// =============================================================================
// 02_DataBlocks.scl
// All non-recipe data blocks.
// Recipe program DBs (DB_RecipeProgram1..10) are in 02b_RecipePrograms.scl.
// They live in LOAD memory; the machine runs from DB_SelectedRecipe (this file).
// Target: CPU 1214C (100KB work memory)
// =============================================================================

// -----------------------------------------------------------------------------
// DB_HMI - Human Machine Interface data
// -----------------------------------------------------------------------------
DATA_BLOCK "DB_HMI"
{ S7_Optimized_Access := 'TRUE' }
VERSION : 0.3
NON_RETAIN
    VAR
        // ===========================================================
        // BUTTONS (Input) - Version_GCODE compatible
        // ===========================================================
        Btn_Start : Bool;           // Start machine
        Btn_Stop : Bool;            // Stop machine
        Btn_Pause : Bool;           // Pause/Resume toggle
        Btn_Reset : Bool;           // Reset program to beginning
        Btn_ApplyToolConfig : Bool;  // Apply tool-slot codes from HMI to DB_ToolConfig
        Btn_AckError : Bool;        // Acknowledge error → transitions from STATE_ERROR to STOPPED
        Btn_Continue : Bool;        // Continue from pause (PAUSED) -- STATE_PAUSED → RUNNING
        Btn_Restart : Bool;         // STATE_ERROR or PAUSED → STOPPED (restart with Start)
        Btn_ProdReset : Bool;       // Reset production counters + history
        Btn_LastCycleReset : Bool;  // Reset last cycle summary only (counters preserved)
                                    // NOTE: Btn_ProdReset already does this too.
                                    // If not adding both as separate HMI buttons, Btn_LastCycleReset
                                    // is redundant -- do not connect to HMI if unused.

        // ===========================================================
        // MODE SELECTION (Input)
        // ===========================================================
        ProductSelect : Int := 1;           // Recipe selector (1-50) -- 50 slots since 2026-08-10 (was 10)
        FeedrateOverride : Real := 100.0;   // Speed % for G1 moves (50-200, 100=normal)
        RapidOverride : Real := 100.0;      // Speed % for G0 rapid moves (50-200)
        SingleStepMode : Bool := FALSE;     // TRUE = stop after each line, wait for StepNext
        StepNext : Bool := FALSE;           // Pulse to advance one step in SingleStepMode

        // Program names and validity.
        //
        // *** DELIBERATELY NOT EXTENDED TO 50 (2026-08-10). Read before touching. ***
        // Verified 2026-08-10: NOTHING in this project writes or reads either array --
        // not the PLC, and not the CAM post-processor (grep gcodes/ for ProgramNames:
        // no hits). They have been declared-and-unused since 1..5. At 50 slots they would
        // cost ~1.1 KB of the 100 KB work memory to stay just as unused, on a CPU that ran
        // out of work memory on 2026-07-31.
        //
        // The name problem is solved two other ways instead:
        //   - WHICH program is loaded now: DB_HMI.LoadedProgramName, a continuous mirror of
        //     DB_SelectedRecipe.Header.sName. One String[20] regardless of slot count.
        //   - BROWSING all 50 names before selection: a WinCC text list keyed off
        //     ProductSelect. Zero PLC bytes, and operator-editable on the HMI, which is what
        //     "operator-defined names" wanted in the first place.
        //
        // Kept at 1..10 rather than deleted because the WinCC project may write them and it
        // is not visible from here -- deleting would silently break an HMI tag connection.
        // If the HMI does not use them either, they are ~230 B of reclaimable work memory.
        ProgramNames : Array[1..10] of String[20];  // UNUSED -- see note above
        ProgramValid : Array[1..10] of Bool;        // UNUSED -- see note above

        // Name of the recipe currently in DB_SelectedRecipe (2026-08-10). PLC-written,
        // read-only for the HMI. Continuous mirror of DB_SelectedRecipe.Header.sName,
        // written at the bottom of FB_Process next to the DB_Diagnostic mirrors -- so it
        // appears in no reset path by design (nothing to clear; it always reports the
        // buffer's true content, blank when the buffer is poisoned or a load failed).
        // 22 bytes, flat regardless of slot count. Display it beside ProductSelect so the
        // operator sees WHICH program is about to run, not just a slot number out of 50.
        // NOTE: CAM currently emits the same generic sName ('SpinningCam Program') for
        // every program -- ask SpinningCam for a distinct name per program or this reads
        // identically for all 50 slots.
        LoadedProgramName : String[20];

        // Recipe checksum pair, PLC-written, read-only for the HMI (2026-08-14).
        // Continuous mirrors written next to LoadedProgramName at the bottom of
        // FB_Process -- in no reset path by design, because they always report the
        // buffer's true state. 9 bytes total.
        //
        // Display these two side by side on the diagnostics screen. They matter only
        // when they DISAGREE, and then they answer the one question 16#0316 cannot:
        // which side is wrong. Three implementations of the algorithm exist
        // (SpinningCam's, tools/split_recipe_db.py, FB_RecipeLoader) and only the
        // first two have ever been checked against each other. If _Calculated is a
        // stable, repeatable number that simply is not _Recipe, suspect the SCL, not
        // the recipe file -- re-exporting a good file will not help and wastes a trip.
        // If _Calculated changes between attempts on the same recipe, the transfer is
        // landing different data each time, which is the original fault.
        //
        // _Verified = TRUE means checked AND matched. FALSE also means "this recipe
        // carries no checksum", so it is not a fault indicator on its own -- a blank
        // _Recipe (0) with _Verified FALSE is a pre-2026-08-14 export loading normally.
        Checksum_Recipe : UDInt;        // what the recipe file declares
        Checksum_Calculated : UDInt;    // what the PLC computed after reassembly
        Checksum_Verified : Bool;       // TRUE = checked and matched


        // Tool slot codes editable from HMI. Enter external codes like 101, 406 etc.
        // These are copied to DB_ToolConfig.ToolCode_List when operator presses Apply.
        ToolSlotCode : Array[1..4] of Int := [101, 102, 103, 104];

        // ===========================================================
        // POSITION DISPLAYS (Output)
        // ===========================================================
        ActualX : Real;             // Current X position (mm)
        ActualZ : Real;             // Current Z position (mm)

        // ===========================================================
        // STATUS DISPLAYS (Output)
        // ===========================================================
        StatusMsg : String[50];     // Status message text
        MachineState : Int;         // State machine state
        CurrentLine : Int;          // Current line being executed
        TotalLines : Int;           // Total lines in program
        // -----------------------------------------------------------
        // Pass display -- mirrored from FB_RecipeHandler every scan.
        // Fed by the CMD=50 / CMD=51 marker lines SpinningCam emits when its
        // PLC-mode "pass markers" option is on. 0 = NO PASS INFORMATION (recipe
        // has no markers, or the first one has not been reached yet), so the HMI
        // must blank the whole group on 0 rather than display "Pass 0 / 0".
        // "Line 47 of 99" means nothing to an operator; "Op 1, pass 3 of 10" is
        // how the job is actually described. See letter_spinningcam_pass_markers.md.
        // -----------------------------------------------------------
        CurrentOp : Int;            // Operation number of the current line (0 = unknown)
        TotalOps : Int;             // Operations in the loaded program (0 = unknown)
        CurrentPass : Int;          // Pass number within the current operation (0 = unknown)
        TotalPasses : Int;          // Passes in the current operation (0 = unknown)
        ProgressPercent : Real;     // Progress 0-100%
        CurrentTool : Int;          // Active tool (1-4)
        FeedrateActive : Real;      // Actual feedrate (mm/min)
        // ⚠️ UNUSED: PLC code does not write to the Axis_Status_* tags below anywhere.
        // They will always be 0 / empty if connected to HMI. Reserved for future use
        // -- do not display on HMI for now.
        Axis_Status_X        : Int;
        Axis_Status_Z        : Int;
        Axis_Status_Spindle  : Int;
        Axis_Status_Toolhead : Int;
        Axis_Status_X_Str        : String[10];
        Axis_Status_Z_Str        : String[10];
        Axis_Status_Spindle_Str  : String[10];
        Axis_Status_Toolhead_Str : String[10];
        // ===========================================================
        // STATUS LAMPS (Output)
        // ===========================================================
        IsRunning : Bool;           // Machine is running
        IsPaused : Bool;            // Machine is paused
        HasError : Bool;            // Error is active
        ElapsedTime : Time;         // Program elapsed time
        ElapsedSeconds : DInt;      // Elapsed time in seconds (for HMI display)
        // CycleCount DELETED 2026-08-15 -- it duplicated "DB_Production".TotalOK and was
        // wrong (its one-shot only cleared on a hard reset, so it counted once per Reset
        // press, not once per part). Parts counting lives in DB_Production alone:
        // TotalStarted / TotalOK / TotalNOK / TotalStopped / TotalAborted. Do not add a
        // parts counter back into DB_HMI.

        // ===========================================================
        // ERROR DISPLAY (Output)
        // ===========================================================
        ErrorID : Word;             // Error code (0=OK)
        ErrorText : String[100];     // Error description
        ErrorDetail : String[120];   // Additional error info

        // ===========================================================
        // WARNING DISPLAY (Output)
        // ===========================================================
        HasWarning : Bool;          // TRUE when a non-blocking warning is active (E-Stop bypass or sheet insert prompt)
        // Key for the HMI's warning text list (ITEM-55). Written every scan next to
        // WarningText, so it needs no reset-path entry: the ELSE branch of the warning
        // block drives it to 0 unconditionally. 0 must stay "no warning".
        //   1 = DANGER: E-Stop bypassed - machine runs unguarded (auto run IS permitted
        //       since 2026-08-12 -- this is the only on-screen sign of it)
        //   2 = Insert sheet, then press both start buttons
        //   3 = Tool axis locked - ToolHeadLock is engaged (manual jog/move/home
        //       on the tool axis refused; see the interlock in FB_Process)
        WarningID : Int;
        WarningText : String[70];   // Warning message text -- English (E-Stop bypass or operator prompts only)
        ResumeLine : Int := -1;     // Saved recipe line for warm restart (-1 = none). Set in STATE_ERROR, cleared on Btn_Restart.

        // End-of-program sanding dwell in progress (2026-08-29). PLC-written, read-only
        // for the HMI. TRUE = the program has finished AND the spindle has been deliberately
        // restarted at DB_MachineConfig.SandSpeed so the operator can sand the part.
        //
        // Display this prominently. MachineState is 100 ('Program Complete') throughout the
        // dwell, so without this flag the screen says the machine is finished while the
        // spindle is turning -- which is exactly the moment an operator reaches in.
        // It is the key for the sanding banner in the WinCC text lists; MachineState cannot
        // serve, because it does not change when the dwell starts or ends.
        //
        // No reset-path entry needed: it is a continuous mirror of the FB_Process latch,
        // written every scan next to the DB_Diagnostic mirrors at the bottom of FB_Process,
        // so it follows the latch to FALSE on every exit path.
        SandActive : Bool;

        // ===========================================================
        // SPANISH TEXT MIRRORS -- REMOVED 2026-08-10 (ITEM-55, stage 1).
        // StatusMsg_ES / ErrorText_ES / ErrorDetail_ES / WarningText_ES are gone,
        // along with the 161 PLC assignments that filled them (~4.9 KB of string
        // literals plus the copy code, on a CPU that hit 101% work memory).
        // Spanish now comes from WinCC text lists keyed off tags the PLC already
        // writes: ErrorID, MachineState, DB_Manual.MDI_Status, and WarningID.
        // The wording was extracted to tools/hmi_texts.csv BEFORE deletion -- use
        // that to populate the text lists; do not retype or re-translate.
        // Do NOT re-add per-language string fields here: each new language then
        // costs work memory again, which is exactly what this removed.
        // ===========================================================

        // ===========================================================
        // BYPASS SWITCHES (for testing) - Version_GCODE compatible
        // ⚠️ All bypasses reset to FALSE on restart (FC_LoadConfig).
        // All must be FALSE in production.
        // ===========================================================
        // ⚠️ Bypass_EStop PERMITS AUTO RUN since 2026-08-12 (it used to block it).
        // The machine will execute a recipe with the E-Stop circuit defeated.
        // Protect this tag with a WinCC user authorization (service login only) --
        // the PLC deliberately no longer second-guesses it. Still forced FALSE by
        // FC_LoadConfig on every power-up, so it cannot survive a restart.
        Bypass_EStop        : Bool := FALSE;  // Used in FB_SafetyMonitor ✅
        Bypass_Door         : Bool := TRUE;  // Used in FB_SafetyMonitor ✅
        Bypass_AirPressure  : Bool := TRUE;  // Used in FB_SafetyMonitor ✅
        Bypass_Drives       : Bool := FALSE;  // Used in FB_SafetyMonitor ✅
        Bypass_Spindle      : Bool := FALSE;  // Skips spindle commands in recipe (FB_RecipeHandler) -- dry run / commissioning
        Bypass_ToolChanger  : Bool := FALSE;  // ⚠️ UNUSED -- not in safety monitor
        // Bypass_MandrelLock DELETED from DB_HMI 2026-08-16 -- it was an ORPHAN. ITEM-33 declared
        // it here as well as in DB_MachineConfig, but every one of the nine read sites, and
        // FC_LoadConfig, use "DB_MachineConfig".Bypass_MandrelLock. This copy was written by
        // nothing and read by nothing. Two identically-named flags where only one is live is a
        // trap: an HMI switch bound to this one would appear to bypass the cylinder and do
        // absolutely nothing. The live flag is DB_MachineConfig.Bypass_MandrelLock -- use that.
        Bypass_ToolHeadLock : Bool := FALSE;  // TRUE = skip ToolHeadLock sensor wait in STATE_LOCK_EXTEND_WAIT (no cylinder/sensor); cylinder still commanded if present
        // A Sim_HomeInPlace flag was added here on 2026-09-06 and REVERTED the same day.
        // It selected MC_Home Mode 0 so a homing cycle could finish in PLCSIM. It cannot
        // work: S7-PLCSIM does not simulate S7-1200 motion control at all -- the
        // technology objects download, but their logic never runs and the PTO hardware is
        // not simulated -- so MC_Power never reports Status and MC_Home never completes,
        // in any mode. Do not re-add it. Nothing past STATE_STARTING can be simulated;
        // what CAN be tested offline is everything before it (recipe load, checksum,
        // pre-scan). See CLAUDE.md and the PLCSIM section of Human_TODO.md.

        // ===========================================================
        // BOUNDING BOX (Output - from pre-scan)
        // ===========================================================
        BoundingBox_MinX : Real;
        BoundingBox_MaxX : Real;
        BoundingBox_MinZ : Real;
        BoundingBox_MaxZ : Real;
        BoundingBox_Valid : Bool;
        PreScanProgress : Real := 0.0;  // Pre-scan progress 0-100% (written during STATE_PRE_SCAN)

        // ===========================================================
        // MANUAL > MANAGE: Contactor & Enable controls (Input)
        // HMI writes these; PLC drives physical outputs in OB1.
        // Buttons are toggles (maintained, not momentary).
        // ===========================================================
        Btn_Contactor_X       : Bool;   // Energize X driver contactor
        Btn_Contactor_Z       : Bool;   // Energize Z driver contactor
        Btn_Contactor_Tool    : Bool;   // Energize Tool driver contactor
        Btn_Contactor_Spindle : Bool;   // Energize Spindle driver contactor
        Btn_Enable_X          : Bool;   // Send enable signal to X drive
        Btn_Enable_Z          : Bool;   // Send enable signal to Z drive
        // Btn_Enable_Tool (2026-08-16): treated exactly like Btn_Enable_X/Z -- an HMI toggle on
        // MANUAL > MANAGE, ALSO forced TRUE by STATE_STARTING on every auto start. Same drive
        // model, same treatment, no settle delay, no bypass term (FC_ContactorControl ANDs the
        // output with Btn_Contactor_Tool). Before this the tool had no enable output at all:
        // the drive's enable was linked on locally, so the servo came up enabled the instant its
        // contactor closed. The wire is now landed on %Q8.1 and that link is removed.
        Btn_Enable_Tool       : Bool;   // Send enable signal to Tool drive

        // MANUAL > MANAGE: Status feedback (Output) for HMI lamps
        // PLC writes these back after applying safety interlock.
        Contactor_X_On       : Bool;
        Contactor_Z_On       : Bool;
        Contactor_Tool_On    : Bool;
        Contactor_Spindle_On : Bool;
        Enable_X_On          : Bool;
        Enable_Z_On          : Bool;
        Enable_Tool_On       : Bool;

        // ===========================================================
        // E-STOP DUAL CHANNEL STATUS (Output - PLC writes, HMI reads)
        // ===========================================================
        EStop_Ch1_OK      : Bool;   // Channel 1 contact state (TRUE=closed=safe)
        EStop_Ch2_OK      : Bool;   // Channel 2 contact state (TRUE=closed=safe)
        EStop_Discrepancy : Bool;   // Ch1 ≠ Ch2 → contact fault, service required
    END_VAR
BEGIN
END_DATA_BLOCK

// -----------------------------------------------------------------------------
// DB_MachineConfig - Machine configuration parameters
//
// RETENTIVITY (changed 2026-08-09) -- NON_RETAIN was REMOVED from this block.
//
// Why: the commissioning values the operator types on the HMI and that FC_LoadConfig
// deliberately does NOT rewrite -- SheetLoadPos_X, SheetLoadPos_Z, SheetLoadTol -- were
// lost on every power cycle. A non-retentive DB is re-initialised from its start values
// in load memory on restart, so the machine came back parking at 200.0 / 170.0 no matter
// what was set on the HMI.
//
// MANUAL STEP REQUIRED IN TIA PORTAL AFTER IMPORTING THIS SOURCE:
//   Open DB_MachineConfig and tick "Retain" on -- at minimum --
//       SheetLoadPos_X, SheetLoadPos_Z, SheetLoadTol, SandTime_s, SandSpeed
//   The other operator-owned values have the same problem and are worth ticking too:
//       SoftLimit_MinX/MaxX/MinZ/MaxZ, SafePos_X/Z, PauseRetract_X/Z/Vel,
//       HomeOffset_X/Z
//   Source import cannot set per-tag retentivity; removing NON_RETAIN only makes the
//   checkbox available. VERIFY the checkboxes after every re-import of this file.
//
//   Do NOT tick Retain on anything FC_LoadConfig writes -- OB100 overwrites it on every
//   restart, so Retain has no effect there and only consumes retentive memory. That is
//   the whole "FIXED" section below, plus these four from the HMI-editable group:
//       HomeVelocity, PostHome_Clearance, AlwaysHomeOnAutoStart, and DB_Manual.HomingMode
//
// NOTE: changing retentivity forces a full re-initialisation of this DB on the next
// download (values return to the start values below). Re-enter the park position on the
// HMI once after that download.
// -----------------------------------------------------------------------------
DATA_BLOCK "DB_MachineConfig"
{ S7_Optimized_Access := 'TRUE' }
VERSION : 0.3
    VAR
        // =====================================================================
        // HMI-EDITABLE: Machine Physical Limits (mm)
        // These values are NOT overwritten by FC_LoadConfig.
        // Can be changed from HMI Setup screen. They survive a PLC restart ONLY if the
        // tag is marked Retain in the TIA DB editor -- see the block header.
        // =====================================================================
        SoftLimit_MinX : Real := -30.0;     // X minimum (home=0)
        SoftLimit_MaxX : Real := 500.0;   // X maximum travel (mm)
        SoftLimit_MinZ : Real := -50.0;  // Z minimum (negative = mandrel front / clearance)
        SoftLimit_MaxZ : Real := 500.0;   // Z maximum (forming depth)

        // HMI-EDITABLE: Safe Positions (mm)
        SafePos_X : Real := 0.0;         // "Go Safe" X target
        SafePos_Z : Real := 0.0;        // "Go Safe" Z target (clearance zone)

        // HMI-EDITABLE: Sheet-Load Park Position (mm)
        // The single position the machine parks at whenever it is waiting for the
        // operator to load a sheet. Reached at the end of every program (STATE_COMPLETE
        // is not used -- the park move is the STOPPING/POST_HOME_CLR path), after every
        // homing cycle, and after a Stop. STATE_STARTING compares the live axis position
        // against it to decide whether the homing seek can be skipped (fast cycle mode).
        //
        // SAFETY: this is where the operator reaches in to insert a sheet and where the
        // MandrelLock clamps. Set it only to a position where the tool head does not
        // obstruct loading. Commission conservatively (near 0,0) and walk it in.
        // Targets are clamped to SoftLimit_Min/Max before any move is issued.
        //
        // Deliberately NOT written by FC_LoadConfig, so OB100 does not fight the HMI.
        // MUST be marked Retain in the TIA DB editor -- see the block header. Without the
        // Retain tick these three revert to the start values below on every power cycle.
        SheetLoadPos_X : Real := 200.0;    // Sheet-load park X target (mm)
        SheetLoadPos_Z : Real := 170.0;    // Sheet-load park Z target (mm)
        SheetLoadTol   : Real := 2.0;    // +/- window counted as "at the park position" (mm)

        // HMI-EDITABLE: Pause Retract (mm / mm/s)
        // On Pause, X and Z jog by these signed offsets to pull the tool clear
        // (spindle keeps running). On Continue they return to the exact interruption
        // point before the recipe resumes. Retract target is clamped to soft limits.
        // Offset 0 = that axis does not move on pause. See docs/FB_Process_States.md
        // (STATE_PAUSED) for the full pause/resume sequence.
        PauseRetract_X   : Real := -10.0;   // Pause retract offset X (signed, mm)
        PauseRetract_Z   : Real := -10.0;   // Pause retract offset Z (signed, mm)
        PauseRetract_Vel : Real := 20.0;    // Retract/return velocity (mm/s)

        // HMI-EDITABLE: Homing Parameters
        HomeOffset_X : Real := 0.0;       // X set value after homing
        HomeOffset_Z : Real := 0.0;       // Z set value after homing
        HomeVelocity : Real := 10.0;      // Homing clearance velocity (mm/s)
        PostHome_Clearance : Real := 10.0; // Distance to clear PNP zone after homing (mm)
        // HMI-EDITABLE: fast cycle mode master switch.
        //   TRUE  = home all axes on every auto start (legacy behaviour)
        //   FALSE = skip the reference seek when the reference is trusted AND the axes
        //           are parked at SheetLoadPos (see FB_Process STATE_STARTING)
        // This switch can only ever skip homing in the NORMAL case. It never overrides
        // FB_Process bRequireHoming -- an E-Stop, a fault or a power-up always re-homes.
        AlwaysHomeOnAutoStart : Bool := FALSE;

        // ⚠️ UNUSED: The following two parameters are not read anywhere in PLC code.
        // Recipe handler takes its own feedrate from the recipe line.
        // Do not connect to HMI. May be used if manual tool change sequence is added later.
        ToolChangePos_X : Real := 0.0;   // (Unused) Safe X for manual tool change
        ToolChangePos_Z : Real := 0.0;  // (Unused) Safe Z for manual tool change
        DefaultFeedrate : Real := 100.0;  // (Unused) Default feedrate

        // =====================================================================
        // FIXED: Hardware/TO Limits -- must not be changed from HMI
        // FC_LoadConfig (OB100) writes these values on every restart.
        // =====================================================================
        MaxVelocity : Real := 40.0;     // mm/s - TO max velocity
        RapidVelocity : Real := 40.0;   // mm/s - G0 rapid speed
        MinVelocity : Real := 1.0;      // mm/s - TO minimum
        FeedrateConvFactor : Real := 60.0; // divisor to convert recipe F (mm/min) to axis velocity (mm/s)

        // EXPERIMENTAL -- velocity-mode continuous path (branch exp/velocity-path-350).
        // VelPath_Enable and VelPath_LeadTime are written by FC_LoadConfig on every
        // restart, so an online change lasts until the next power cycle. VelPath_Enable
        // is forced FALSE there -- the experiment must be switched on deliberately.
        // VelPath_MaxDeviation is OPERATOR-OWNED (2026-09-16): HMI-editable, NOT written
        // by FC_LoadConfig, needs a manual Retain tick (docs/RETAINED_TAGS.md). Without
        // the tick it falls back to the start value below at power-up.
        // Design and test plan: docs/MotionSmoothing.md section 9.
        VelPath_Enable       : Bool := TRUE; // TRUE = runs of G1 lines use MC_MoveVelocity (no stop per line)
        VelPath_LeadTime     : Real := 0.09;   // s -- next line takes over at feed x this before the end point (capped at half the segment). Tuned with the jerk-aware sim (scan 45 ms, t1 0.06)
        VelPath_MaxDeviation : Real := 2.0;   // mm -- HMI-EDITABLE. Start value raised 1.0 -> 2.0 on 2026-09-21 (user). Off-path / backwards distance that faults with 16#000F. PLC clamps to 0.05..5.0 (VM_MAXDEV_MIN/MAX in 05_RecipeHandler.scl -- the clamped value is what the fault text prints). Above 0.8 mm (the final-pass roller-mandrel gap = sheet thickness) it no longer protects the mandrel

        // Tool Configuration -- HMI-EDITABLE: active slot count (1-4)
        ToolCount    : Int  := 3;
        ToolVelocity : Real := 50.0;   // deg/s -- turret rotation speed (clamped by TO max)

        // Hardware configuration -- set TRUE if this axis is not physically connected to the machine
        // (different from HMI bypasses: this is a hardware presence flag)
        Bypass_ToolAxis : Bool := FALSE;
        // THE live MandrelLock bypass -- all nine read sites and FC_LoadConfig use this one.
        // (A duplicate in DB_HMI was deleted 2026-08-16; it was never read.)
        // TRUE = no MandrelLock cylinder, sheet clamped manually. FC_LoadConfig sets the
        // per-machine value on every power-up and overrides this start value -- change it there,
        // not here. On THIS machine it is TRUE.
        Bypass_MandrelLock : Bool := FALSE;
        // Spindle deceleration wait: time between RunCmd=FALSE and next RunCmd=TRUE.
        // Set to match VFD deceleration ramp time. HMI-editable.
        SpindleDecelTime : Time := T#2S;
        // Pause resume spin-up wait: on Continue from PAUSED, the spindle is
        // restarted and this time is allowed for it to ramp back up to speed
        // BEFORE the axes return to the interruption point and machining resumes.
        // The axes stay clear of the workpiece (held at the pause-retract position)
        // for this whole window. Set to the measured VFD ramp-up time + margin.
        SpindleResumeSpeedupTime : Time := T#5S;
        // Load-memory recipe copy (FB_RecipeLoader, STATE_RECIPE_LOAD(11)):
        // hang watchdog on the READ_DBL transfer. A 1000-line recipe is ~12 KB
        // and completes in well under a second; this only catches a transfer
        // that never reports BUSY=FALSE. Expiry -> 16#0312, machine goes to
        // STATE_ERROR rather than starting a cycle on a half-copied recipe.
        RecipeLoadTimeout : Time := T#10S;
        // In-place spindle speed change (FB_SpindleControl): how long MC_MoveVelocity
        // Execute is held LOW to regenerate the trigger edge for the new velocity.
        // RunForward (VFD run) stays TRUE throughout -- only the PTO command edge is
        // regenerated. T#0S = one PLC scan. Increase if the VFD needs more settle
        // time before the new velocity command. Tune on-site.
        SpindleSpeedChange_ExecLowTime : Time := T#0S;
        // Speed-change mode selector (VFD-dependent -- confirm on the bench):
        //   FALSE = keep RunForward TRUE during the change (VFD tracks pulse-train
        //           frequency live; this is the documented wiring intent).
        //   TRUE  = also drop RunForward during the Execute-low window, then re-assert
        //           it. Use only if the drive latches its frequency at the RunForward
        //           rising edge and ignores a live frequency change. Safe re: PTO --
        //           the pulse train keeps running; RunForward is the stop signal.
        SpindleSpeedChange_DropRunForward : Bool := FALSE;
        // Proportional MandrelLock release wait (ITEM-28).
        // SpindleStopSafeTime = full-speed stop safety margin (tune to measured VFD decel time + margin).
        // Formula: PT = (capturedRPM / SpindleMaxRPM) * SpindleStopSafeTime
        // NOT a speed limit -- the only spindle limit is DB_Spindle.MaxSpeed (3000). This is the
        // denominator that scales the coast-down wait, and 2400 is deliberately BELOW it:
        // a smaller denominator makes PT longer, so the MandrelLock waits a little more than
        // strictly needed before releasing. Do NOT "sync" this to DB_Spindle.MaxSpeed -- raising
        // it to 3000 SHORTENS a safety wait. (An older comment here said "match
        // DB_Spindle.MaxSpeed"; that was misleading and is why this note exists. 2026-08-16.)
        SpindleMaxRPM       : Real := 2400.0;  // RPM -- denominator for the proportional wait only
        SpindleStopSafeTime : Time := T#20S;   // Full-speed decel safety margin (tune on-site)

        // ─── HMI-EDITABLE: End-of-program sanding dwell (2026-08-29)
        // After a program finishes, STATE_COMPLETE(100) restarts the spindle at SandSpeed
        // and holds it for SandTime_s seconds so the operator can sand the part before removing it.
        //
        // WHY IT IS A RESTART AND NOT A "KEEP RUNNING": by the time the machine reaches
        // STATE_COMPLETE the spindle is already fully stopped, and it cannot be otherwise.
        // The CAM emits CMD=21 (Spindle OFF) as the second-to-last recipe line, and
        // FB_RecipeHandler STATE_SPINDLE_STOP_WAIT(58) BLOCKS on DB_Spindle.IsRunning=FALSE
        // before it will advance to the CMD=99 END marker. So the dwell necessarily begins
        // after a stop, and costs the VFD's ramp-down + ramp-up (~2 s) before the part turns
        // again. Do not "optimise" that away by suppressing the final CMD=21 -- a recipe has
        // several CMD=21 lines (program 1 has four: 51, 60, 69, 70) and picking the right one
        // needs a pre-scan pass whose failure mode is a spindle left running.
        //
        // BOTH must be > 0 for the dwell to arm. SandTime_s := 0 (the download default)
        // is the OFF switch and leaves end-of-program behaviour exactly as it was.
        //
        // UNITS: SandTime_s is WHOLE SECONDS as a plain Int -- deliberately NOT the Time
        // type every other timer in this DB uses. An S7 Time is milliseconds underneath,
        // so an operator typing "10" into a numeric field would get 10 ms and conclude the
        // feature is broken. The other timers are commissioning values a technician sets
        // once from the TIA editor; this one is retyped at the machine per job, so the
        // units have to survive a plain number field. FB_Process clamps it to
        // 0..SAND_TIME_MAX_S (600 s) and converts to a Time PT.
        //
        // SAFETY: this is the one feature that invites a hand near a turning part. The door
        // interlock does NOT protect it -- FC_LoadConfig forces Bypass_Door := TRUE on every
        // power-up on this machine. What does stop it: E-Stop (drops bDrivesEnable, which is
        // FB_SpindleControl's Enable) and the Stop button (STATE_COMPLETE is excluded from
        // the STOPPING path, so Stop goes straight to STOPPED and STOPPED clears the spindle).
        // Commission SandSpeed LOW -- it is a hand-sanding speed, not a cutting speed.
        //
        // Deliberately NOT written by FC_LoadConfig, so OB100 does not fight the HMI.
        // MUST be marked Retain in the TIA DB editor -- see the block header. Without the
        // Retain tick these two revert to the start values below on every power cycle.
        SandTime_s : Int  := 0;        // SECONDS. 0 = feature off. Spindle run time at end of program. Clamped 0..600.
        SandSpeed  : Real := 0.0;      // RPM during the dwell. Clamped to DB_Spindle.MinSpeed/MaxSpeed.

        // ─── Cylinder stroke wait times (open-loop: tuned to physical stroke duration)
        // These are deliberate waits with no sensor feedback. Set slightly above measured stroke time.
        CylMandrelLock_ClampTime    : Time := T#5S;    // STATE_SHEET_WAIT ph.2: MandrelLock clamp stroke
        CylSheetHolder_RetractTime  : Time := T#5S;    // STATE_SHEET_WAIT ph.3: SheetHolder retract stroke
        CylToolHeadLock_PreDelay    : Time := T#1S;    // STATE_LOCK_EXTEND_WAIT: pre-delay before solenoid energises
        CylToolHeadLock_RetractTime : Time := T#3S;    // STATE_LOCK_RETRACT_WAIT: spring-return wait (no sensor)
        CylBackSupport_EndRetractTime : Time := T#2S;  // End-of-recipe BackSupport retract: Sol_B held this long, then all coils off

        // ─── Process timeouts (trigger errors when limits exceeded)
        Timeout_DriveReady     : Time := T#3S;     // STATE_STARTING: drives not ready within this time → error
        // NOTE: there is deliberately no tool-enable settle delay. The tool servo is the same
        // drive as X and Z, which assert enable in the same scan as their contactor and have
        // always worked. See STATE_STARTING in 06_MainProcess.scl.
        Timeout_Homing         : Time := T#120S;   // STATE_HOMING + STATE_STOP_GOHOME combined timeout
        Timeout_Motion         : Time := T#300S;   // Per-line G0/G1 motion timeout in FB_RecipeHandler
        Timeout_SpindleAtSpeed : Time := T#10S;    // CMD=20: spindle must reach target speed within this time
        Timeout_SpindleStop    : Time := T#15S;    // CMD=21: spindle must reach zero within this time
        Timeout_ToolChange     : Time := T#30S;    // Turret rotation must complete within this time
        Timeout_EStopDiscrep   : Time := T#500MS;  // E-Stop dual-channel discrepancy debounce
    END_VAR
BEGIN
END_DATA_BLOCK

// DB_ErrorCodes removed -- error codes are used as inline hex constants.
// Severity: 0=info, 1=warn, 2=error, 3=fatal

// -----------------------------------------------------------------------------
// DB_Error - Centralized error snapshot for debugging (non-invasive to HMI)
// -----------------------------------------------------------------------------
DATA_BLOCK "DB_Error"
{ S7_Optimized_Access := 'TRUE' }
VERSION : 0.1
NON_RETAIN
    VAR
        Active    : Bool := FALSE;       // TRUE when an active error is present
        Code      : Word := 0;           // Error code (matches DB_ErrorCodes)
        Severity  : Byte := 0;           // Priority tier: 1=warning, 2=project, 3=motion/TO, 4=safety (higher preempts lower on HMI display)
        Source    : String[20];          // Originating FB or category (e.g. 'Recipe', 'Safety')
        Line      : Int := -1;           // Recipe line (if applicable) or -1
        TimeStamp : DTL;                 // Timestamp captured with RD_SYS_T
        Details   : String[120];          // Free text details / ActiveErrorText
        // History ring buffer (last 10 errors) for post-mortem analysis
        History_Code    : Array[1..10] of Word;
        History_Time    : Array[1..10] of DTL;
        History_Source  : Array[1..10] of String[20];
        // String[40] (was String[80], 2026-07-31 memory reclaim -- saves 400 B).
        // Matches AlarmEntry.ErrorText[40] in DB_AlarmHistory, so both history views
        // truncate identically. Written via LEFT(..., 40) in FB_AlarmManager.
        History_Details : Array[1..10] of String[40];
        History_Index   : Int := 0;      // 1..10
        History_Count   : Int := 0;      // Number of valid entries (<=10)
        TotalErrorCount : DInt := 0;     // Lifetime error count (incremented on each new error)
    END_VAR
BEGIN
END_DATA_BLOCK

// -----------------------------------------------------------------------------
// DB_ToolConfig - Tool changer configuration
// -----------------------------------------------------------------------------
DATA_BLOCK "DB_ToolConfig"
{ S7_Optimized_Access := 'TRUE' }
VERSION : 0.2
NON_RETAIN
    VAR
        // Slot angles -- automatically calculated by FC_ToolAngleCalc (AutoCalcAngles=TRUE)
        // or manually entered from HMI Tool page (AutoCalcAngles=FALSE).
        // Machine has 3 physical slots: 0 / 120 / 240 deg. Slot 4 is unused (ToolCount=3).
        Tool1_Position : Real := 0.0;     // Slot 1 angle (degrees)
        Tool2_Position : Real := 120.0;   // Slot 2 angle (degrees)
        Tool3_Position : Real := 240.0;   // Slot 3 angle (degrees)
        Tool4_Position : Real := 0.0;     // Slot 4 unused (ToolCount=3)

        // Slot code mapping -- can be entered from HMI Tool page.
        // Operator enters which head code is in which slot.
        ToolCode_List : Array[1..4] of Int := [101, 102, 103, 104];

        CurrentTool : Int := 1;           // Active slot number (1-4)

        // HMI Tool page: automatic angle calculation
        // TRUE = calculate evenly spaced based on ToolCount (3 slots → 0/120/240)
        // FALSE = Tool1..4_Position open for manual entry
        AutoCalcAngles : Bool := TRUE;

        // Calculated step angle -- displayed on HMI for information (e.g. "90°/slot")
        ToolStepAngle_Calc : Real := 120.0;
    END_VAR
BEGIN
END_DATA_BLOCK

// -----------------------------------------------------------------------------
// DB_Spindle - Spindle configuration and status
// -----------------------------------------------------------------------------
DATA_BLOCK "DB_Spindle"
{ S7_Optimized_Access := 'TRUE' }
VERSION : 0.2
NON_RETAIN
    VAR
        // Configuration
        MinSpeed : Real := 120.0;         // Minimum spindle speed (RPM)
        MaxSpeed : Real := 3000.0;        // Maximum spindle speed (RPM)
        DefaultSpeed : Real := 1200.0;    // Default spindle speed (RPM)
        SpeedTolerance : Real := 5.0;     // Speed tolerance for AtSpeed (%)
        Bypass_AtSpeed : Bool := FALSE;   // TRUE = skip AtSpeed wait (use during commissioning without drive)

        // Commands (input from HMI/Program)
        Cmd_SetSpeed : Real;              // Commanded speed
        Cmd_Direction : Int;              // 1=CW, -1=CCW
        SpeedOverride : Real := 100.0;    // Speed override (%)

        // Status (output)
        IsRunning : Bool := FALSE;
        AtSpeed : Bool := FALSE;
        ActualSpeed : Real := 0.0;
        CommandedSpeed : Real := 0.0;
        Error : Bool := FALSE;
        ErrorID : Word := 0;

        // =====================================================================
        // DIAGNOSTICS -- written every scan; read from HMI watch table
        // Use these to trace the spindle start chain without TIA Portal online.
        // Chain:  ReqStart → bSpindleStart → StartInput → PrevStart → StartEdge → state
        // =====================================================================
        Diag_SpindleState  : Int;   // FB_SpindleControl state (0=Idle, 10=Starting, 20=Running, 30=Stopping, 999=Error)
        Diag_StartInput    : Bool;  // Actual Start pin arriving at FB_SpindleControl (Manual OR bSpindleStart)
        Diag_StopInput     : Bool;  // Actual Stop pin arriving at FB_SpindleControl
        Diag_EnableInput   : Bool;  // Actual Enable pin (bDrivesEnable)
        Diag_StartEdge     : Bool;  // Rising edge computed inside FB_SpindleControl (TRUE = spindle command accepted)
        Diag_PrevStart     : Bool;  // prevStart latch inside FB_SpindleControl (must go FALSE between starts)
        Diag_bSpindleStart : Bool;  // FB_Process internal flag bSpindleStart (set by recipe or RUNNING state)
        Diag_bSpindleStop  : Bool;  // FB_Process internal flag bSpindleStop
        Diag_ReqStart      : Bool;
        Diag_ReqStop       : Bool;
        Diag_MoveVelBusy   : Bool;  // MC_MoveVelocity.Busy   -- TO is processing the velocity command
        Diag_MoveVelInVel  : Bool;  // MC_MoveVelocity.InVelocity -- motor reached commanded speed

        // =====================================================================
        // HISTORY RING BUFFER -- last 20 state-change snapshots
        // A new entry is pushed whenever SpindleState, PrevStart, ReqStart or
        // StartEdge changes, capturing every meaningful transition in sequence.
        //
        // How to read:
        //   1. Hist_Count tells you how many valid entries exist (0..20).
        //   2. Hist_Head-1 (mod 20) is the MOST RECENT entry.
        //   3. Entries are indexed [0..19]; read them in Seq order.
        //   4. Write Hist_Clear := TRUE from HMI to wipe and start fresh.
        // =====================================================================
        Hist_Head  : Int := 0;          // Next write position (0..19, wraps)
        Hist_Count : Int := 0;          // Number of valid entries (0..20)
        Hist_SeqNum : Int := 0;         // Rolling sequence counter
        Hist_Clear  : Bool := FALSE;    // HMI: write TRUE to clear buffer (auto-resets)
        Hist_Log   : Array[0..19] of "UDT_SpindleSnap";
    END_VAR
BEGIN
END_DATA_BLOCK

// -----------------------------------------------------------------------------
// DB_Diagnostic - Runtime diagnostics and debugging
// -----------------------------------------------------------------------------
DATA_BLOCK "DB_Diagnostic"
{ S7_Optimized_Access := 'TRUE' }
VERSION : 0.1
NON_RETAIN
    VAR
        // =========================================================
        // PROCESS STATE
        // =========================================================
        Process_State : Int;
        Process_SafeToRun : Bool;
        Process_DrivesEnable : Bool;

        // =========================================================
        // RECIPE HANDLER STATE
        // =========================================================
        Recipe_CurrentProgram : Int;    // Active program number (1-50)
        // Which recipe is actually sitting in DB_SelectedRecipe (0 = none/invalid).
        // Written by STATE_RECIPE_LOAD(11) after a successful READ_DBL copy.
        // Diagnostic value: if this disagrees with Recipe_CurrentProgram, the
        // buffer is stale and the machine would be cutting the wrong geometry.
        Recipe_LoadedProgram : Int;
        Recipe_CurrentLine : Int;       // Current line being executed
        Recipe_TotalLines : Int;        // Total lines in program
        Recipe_TargetX : Real;          // Current target X
        Recipe_TargetZ : Real;          // Current target Z
        Recipe_Velocity : Real;         // Current velocity
        // Pre-scan results
        PreScan_Complete : Bool;
        PreScan_Valid : Bool;           // No limit violations found
        PreScan_ErrorLine : Int;        // Line with limit error (-1 if none)

        // =========================================================
        // MOVE STATUS
        // =========================================================
        MoveX_Busy : Bool;
        MoveX_Done : Bool;
        MoveX_Error : Bool;
        MoveZ_Busy : Bool;
        MoveZ_Done : Bool;
        MoveZ_Error : Bool;
        bMoveX : Bool;                  // X axis needs to move
        bMoveZ : Bool;                  // Z axis needs to move

        // =========================================================
        // AXIS INFO (commissioning)
        // =========================================================
        Axis_X_Pos : Real;
        Axis_Z_Pos : Real;
        Axis_X_Enabled : Bool;
        Axis_Z_Enabled : Bool;
        Axis_X_Homed : Bool;
        Axis_Z_Homed : Bool;
        // FB_Process bRequireHoming: TRUE = reference suspect, next auto start WILL home
        // regardless of AlwaysHomeOnAutoStart. Useful on the HMI to explain to the
        // operator why a cycle homed when fast cycle mode is enabled.
        Require_Homing : Bool;

        // =========================================================
        // ERROR CONTEXT
        // =========================================================
        Error_ProcessState : Int;
        Error_Line : Int;
        Error_Code : Word;
        // TO error codes -- raw WORD codes from Siemens MC_ function blocks.
        // Converted to readable text via FC_TO_ErrorText; compare with TIA Portal TO Diagnostics.
        MoveX_ErrorID  : Word;    // MC_MoveAbsolute X axis TO code
        MoveZ_ErrorID  : Word;    // MC_MoveAbsolute Z axis TO code
        HomeX_ErrorID  : Word;    // MC_Home X axis TO code
        HomeZ_ErrorID    : Word;   // MC_Home Z axis TO code
        HomeTool_ErrorID : Word;  // MC_Home Tool axis TO code
        Power_X_ErrorID : Word;   // MC_Power X axis TO code
        Power_Z_ErrorID : Word;   // MC_Power Z axis TO code
        // Added 2026-08-17. Its absence is why the one axis the alarm named was the one
        // axis whose TO code could not be recovered after the fact -- fbPowerTool.ErrorID
        // is volatile and Reset (MC_Reset) erases it. Latched like X/Z: written whenever
        // MC_Power reports an error, never cleared, so non-zero means "this axis faulted
        // at some point this power cycle".
        Power_Tool_ErrorID : Word; // MC_Power Tool axis TO code
        Spindle_TO_ErrorID : Word; // MC_Power/MC_MoveVelocity/MC_Halt spindle TO code
        Error_Text   : String[100];
        // Error_Detail removed -- not written anywhere, Error_Text is used instead
        // Readable description for the last TO error code (FC_TO_ErrorText output)
        TO_ErrorText : String[60];

        // =========================================================
        // CYLINDER DIAGNOSTICS -- indexed by cylinder number (1-based, max 8)
        // No new fields needed when adding cylinders -- write to CylDiag[N] in OB1.
        // =========================================================
        CylDiag : Array[1..8] of "UDT_CylDiag";
    END_VAR
BEGIN
END_DATA_BLOCK

// -----------------------------------------------------------------------------
// DB_Manual - Manual mode control
// -----------------------------------------------------------------------------
DATA_BLOCK "DB_Manual"
{ S7_Optimized_Access := 'TRUE' }
VERSION : 0.3
NON_RETAIN
    VAR
        ManualModeActive : Bool;
        SelectedAxis : Int := 0;        // 0=X, 1=Z, 2=Tool, 3=Spindle
        ActiveAxis : Int := -1;         // Currently active axis (-1 = none)
        JogSpeed : Real := 10.0;        // mm/s
        JogIncrement : Real := 1.0;     // mm per step
        HomingMode : Int := 3;          // 0=Passive, 2=Active, 3=Active+Zero
        HomePosition : Real := 0.0;     // Home position offset

        // Jog buttons (both naming conventions)
        Btn_JogPlus : Bool;
        Btn_JogMinus : Bool;
        Jog_Plus : Bool;                // Alias
        Jog_Minus : Bool;               // Alias
        Btn_StepPlus : Bool;            // Incremental step +
        Btn_StepMinus : Bool;           // Incremental step -

        // Homing buttons
        Btn_Home : Bool;
        Btn_HomeAxis : Bool;            // Alias for Btn_Home
        Btn_HomeAll : Bool;             // Home all axes
        Btn_GoSafe : Bool;
        Btn_GoZero : Bool;

        // Absolute move
        MoveToPosition : Real := 0.0;   // Target position
        Btn_MoveAbsolute : Bool;        // Execute move

        // Tool step buttons
        Btn_ToolStepCW : Bool;          // Tool step clockwise
        Btn_ToolStepCCW : Bool;         // Tool step counter-clockwise
        ToolStepAngle : Real := 120.0;  // Manual turret step (deg) -- 3 slots at 120 deg spacing
        ToolStepSpeed : Real := 30.0;   // Tool step velocity (deg/s)
        ToolPosition : Real;            // Current tool position (degrees)

        // Spindle manual control
        Btn_SpindleStart : Bool;        // Start spindle
        Btn_SpindleStop : Bool;         // Stop spindle
        Btn_SpindleAckError : Bool;     // Acknowledge spindle error only (machine reset not required)
        Manual_SpindleSpeed : Real := 500.0;  // Spindle speed (RPM)
        Manual_SpindleDir : Int := 1;   // 1=CW, -1=CCW

        // Status (multiple naming conventions for HMI compatibility)
        JogBusy : Bool;
        ManualBusy : Bool;              // Alias for JogBusy
        JogError : Bool;
        ManualError : Bool;             // Alias for JogError
        JogErrorID : Word;
        ManualErrorID : Word;           // Alias for JogErrorID

        // Selected axis info (output)
        SelectedAxisName : String[20];
        SelectedAxisPos : Real;
        SelectedAxisHomed : Bool;
        SelectedAxisReady : Bool;

        // ===========================================================
        // CYLINDER MANUAL CONTROL
        // One HMI screen controls all cylinders via SelectedCylinder.
        // HMI writes to these fields; FC_CylinderDispatch routes to
        // the correct DB_CylinderX instance each scan.
        // To add a cylinder: add DB_CylinderN in 02_DataBlocks.scl,
        // add OB1 calls, and add a CASE branch in FC_CylinderDispatch.
        // ===========================================================
        SelectedCylinder    : Int  := 1;    // Active cylinder (1..N)
        Btn_CylExtend       : Bool;         // Extend command
        Btn_CylExtendFull   : Bool;         // Full extend (ignore sensor)
        Btn_CylRetract      : Bool;         // Retract command
        Btn_CylRetractFull  : Bool;         // Full retract (bypass sensors, pulse use)
        Btn_CylGotoPos      : Bool;         // Rising edge: go to target (Mode 2 = zone-pulse, Mode 3 = extend to level)
        Cyl_TargetPos       : Real := 0.0;  // [Modes 2+3] Target position (mm)
        Cyl_Tolerance       : Real := 2.0;  // [Mode 2] Tolerance written to cylinder DB on Btn_ApplyType press
        Btn_ApplyType       : Bool;         // Rising edge: write SelCyl_SetType + Cyl_Tolerance → cylinder DB
        SelCyl_SetType      : Int  := 0;    // Desired PositioningMode (0–3) — HMI input field
        prevBtn_ApplyType   : Bool;         // Edge detection (internal, not for HMI)

        // ===========================================================
        // MANUAL CMD=40 / CMD=41 (BackSupport)
        // Manual-page equivalents of the recipe commands. Each button
        // writes exactly what the matching recipe line writes.
        // Handled in FB_Process STATE_MANUAL (5) only -- STATE_STOPPED
        // and STATE_ERROR clear all three target flags every scan.
        // ===========================================================
        Btn_Cmd40_Extend    : Bool;         // = CMD=40      : BackSupport extend (level -- hold to extend)
        Btn_Cmd41_AtmoOn    : Bool;         // = CMD=41 P1   : Sol_B override + atmosphere valve ON
        Btn_Cmd41_AtmoOff   : Bool;         // = CMD=41 P2   : atmosphere valve OFF (Sol_B stays ON)
        Btn_Cmd41_Release   : Bool;         // = CMD=41 P3   : release both overrides

        // ===========================================================
        // MANUAL MDI -- type a CMD number + Param and execute it.
        // Generic entry point for auxiliary recipe commands, so a new
        // CMD only needs a CASE branch in FB_Process STATE_MANUAL --
        // no new DB field and no HMI screen change.
        // Motion commands (CMD=0/1) are deliberately NOT accepted here;
        // use Btn_MoveAbsolute for manual positioning.
        // ===========================================================
        MDI_Cmd             : Int;          // Command number to execute (40, 41, ...)
        MDI_Param           : Int;          // Command parameter (meaning depends on MDI_Cmd)
        Btn_MDI_Execute     : Bool;         // Rising edge: execute MDI_Cmd once
        // MDI_Status doubles as the key for the HMI's MDI text list (ITEM-55), so every
        // distinct message needs its OWN value -- 5 and 6 exist only because 1 and 3
        // each used to carry two different messages, which a text list would collapse.
        // 0=idle  1=Executed  2=unknown/blocked CMD  3=CMD40 bad Param
        // 4=CMD40 cylinder error  5=CMD40 done  6=CMD41 bad Param
        MDI_Status          : Int;
        MDI_StatusText      : String[24];   // Result text (EN)
        // MDI_StatusText_ES removed 2026-08-10 (ITEM-55) -- Spanish comes from a
        // WinCC text list keyed off MDI_Status. NOTE: MDI_Status is not yet unique --
        // values 1 and 3 each carry two different messages, so two new values must be
        // assigned before the text list can distinguish them. See tools/hmi_texts.csv
        // (rows marked COLLISION).

        // Selected cylinder status (PLC → HMI)
        SelCyl_Name         : String[20];   // "Cylinder 1" etc.
        SelCyl_State        : Int;          // State code
        SelCyl_StateText    : String[14];   // State text
        SelCyl_AtSetpoint   : Bool;         // Held at setpoint sensor
        SelCyl_AtRetract    : Bool;         // At retract end
        SelCyl_AtTarget     : Bool;         // Ruler mode: within Tolerance
        SelCyl_PosError     : Real;         // Ruler mode: error = actual - target (mm)
        SelCyl_Error        : Bool;         // Active error
        SelCyl_ErrorID      : Word;         // Error code (16#05xx)
        SelCyl_ActualPos    : Real;         // Current position (mm) from analog sensor
        SelCyl_Type         : Int;          // Positioning mode: 0=Full stroke, 1=PNP sensor, 2=Linear ruler
        SelCyl_Toleranse    : Real;         // Position tolerance (mm) - ruler mode only
        SelCyl_MaxPos       : Real;         // Max allowed position (mm) - ruler mode only
        SelCyl_MinPos       : Real;         // Min allowed position (mm) - ruler mode only
    END_VAR
BEGIN
END_DATA_BLOCK

// -----------------------------------------------------------------------------
// DB_HMI_Errors - Error bits + Word triggers for HMI Alarm View
// -----------------------------------------------------------------------------
DATA_BLOCK "DB_HMI_Errors"
{ S7_Optimized_Access := 'TRUE' }
VERSION : 0.1
NON_RETAIN
    VAR
        // Alarm Words (for HMI Discrete Alarm view)
        AlarmWord_Axis : Word;
        AlarmWord_Limits : Word;
        AlarmWord_Tool : Word;
        AlarmWord_Recipe : Word;
        AlarmWord_Safety : Word;
        AlarmWord_Spindle : Word;
        AlarmWord_TO : Word;
        // Individual Bool flags
        Err_X_MoveFailed : Bool;
        Err_Z_MoveFailed : Bool;
        Err_X_HomingFailed : Bool;
        Err_Z_HomingFailed : Bool;
        Err_DriveFault : Bool;
        Err_ToolDrivePower : Bool;  // ITEM-29: tool axis drive power fault (error code 0x000D)
        Err_ToolMoveFailed : Bool;
        Err_ToolHomingFailed : Bool;
        Err_MotionTimeout : Bool;
        Err_LockExtendTimeout : Bool;   // 16#0012 -- ToolHeadLock did not confirm engaged within timeout
        Err_SoftLimit_X_Min : Bool;
        Err_SoftLimit_X_Max : Bool;
        Err_SoftLimit_Z_Min : Bool;
        Err_SoftLimit_Z_Max : Bool;
        Err_HWLimit_X_Min : Bool;
        Err_HWLimit_X_Max : Bool;
        Err_HWLimit_Z_Min : Bool;
        Err_HWLimit_Z_Max : Bool;
        Err_InvalidToolNum : Bool;
        Err_ToolOutOfRange : Bool;
        Err_ToolRotTimeout : Bool;
        Err_ToolRetractFail : Bool;
        Err_ToolRotFailed : Bool;
        Err_Recipe_InvalidCmd : Bool;
        Err_Recipe_ParseErr : Bool;
        Err_Recipe_Empty : Bool;
        Err_Recipe_NoLines : Bool;
        Err_PreScan_Limits : Bool;
        Err_Recipe_Feedrate : Bool;
        Err_Recipe_Timeout : Bool;
        Err_Recipe_ToolNum : Bool;
        Err_EStop : Bool;
        Err_EStop_Discrepancy : Bool;   // E-Stop contact discrepancy (channel fault)
        Err_DoorOpen : Bool;
        Err_DrivesNotReady : Bool;
        Err_AirPressure : Bool;
        Err_SafetyInterlock : Bool;
        Err_Spindle_Power : Bool;
        Err_Spindle_Run : Bool;
        Err_Spindle_Halt : Bool;
        Err_Spindle_Speed : Bool;
        Err_TO_Position : Bool;
        Err_TO_Velocity : Bool;
        Err_TO_NotReady : Bool;
        Err_TO_NotEnabled : Bool;
        Err_TO_LimitExceeded : Bool;
        // Summary flags
        AnyError : Bool;
        AnySafetyError : Bool;
        AnyAxisError : Bool;
        AnyLimitError : Bool;
        AnyToolError : Bool;
        AnyRecipeError : Bool;
        AnySpindleError : Bool;
    END_VAR
BEGIN
END_DATA_BLOCK

// -----------------------------------------------------------------------------
// DB_Production - Production counters and last cycles
// -----------------------------------------------------------------------------
// RETENTIVITY (changed 2026-08-15) -- NON_RETAIN was REMOVED from this block, for the
// same reason it was removed from DB_MachineConfig on 2026-08-09.
//
// A block declared NON_RETAIN is non-retentive as a WHOLE -- the per-tag "Retain"
// checkbox in the TIA DB editor is greyed out. So while that keyword was here, the
// production counters could not be made to survive a power cycle no matter what anyone
// ticked, and "reset every restart" was not a choice anybody made, it was a side effect.
//
// Removing the keyword does NOT make anything retentive. It only makes the tick POSSIBLE.
// The tick is a manual TIA step -- source import cannot set per-tag retentivity -- and it
// must be redone and verified after every re-import of this file. See
// Program/docs/RETAINED_TAGS.md for the full list and the procedure.
//
//   Tick Retain on: TotalStarted, TotalOK, TotalNOK, TotalStopped, TotalAborted
//   Leave alone:    CurrentActive / CurrentProgram / CurrentStartTime (in-flight cycle
//                   state -- a cycle cannot survive a power cycle, and a stale
//                   CurrentActive = TRUE would make the next STOPPED edge count a phantom
//                   abort), and the Last* summary (describes a cycle from before the
//                   restart; harmless either way, but not worth retentive memory).
//
// Changing retentivity forces a full DB re-initialisation on the next download, so the
// counters zero once when this lands. They zeroed on every power cycle before, so nothing
// is lost that was not already being lost.
DATA_BLOCK "DB_Production"
{ S7_Optimized_Access := 'TRUE' }
VERSION : 0.2
    VAR
        // Overall counters.
        // INVARIANT: TotalStarted = TotalOK + TotalNOK + TotalStopped + TotalAborted
        //            + (1 if CurrentActive). Every cycle that starts lands in exactly
        //            one outcome bucket -- see the PRODUCTION LOGGING block in
        //            06_MainProcess.scl. If you add a new way to end a cycle, give it a
        //            bucket there or this stops adding up.
        TotalStarted  : DInt := 0;       // All cycles that entered RECIPE_LOAD (11) -- i.e. every
                                         // accepted Start press. Was PRE_SCAN (12) until 2026-08-15,
                                         // which missed every start that died in the recipe load
                                         // (16#0312 / 16#0314 / 16#0316): not counted as started,
                                         // and not counted as failed either.
        TotalOK       : DInt := 0;       // Completed successfully (STATE=100)
        TotalNOK      : DInt := 0;       // Ended in ERROR (STATE=999)
        TotalStopped  : DInt := 0;       // Operator pressed Stop -- reached STOPPED via the
                                         // STOP sequence (STOPPING / LOCK_RETRACT_WAIT / legacy
                                         // GOHOME / GOTOZERO), so the axes parked cleanly
        TotalAborted  : DInt := 0;       // Cycle ended at STOPPED by any OTHER route -- in practice
                                         // Reset pressed from an active state, which sets
                                         // State := STOPPED directly with no park sequence.
                                         // Added 2026-08-15: these cycles previously hit no bucket
                                         // at all and left CurrentActive stranded TRUE.

        // Current active cycle
        CurrentActive    : Bool := FALSE;
        CurrentProgram   : Int := 0;     // Active program number
        CurrentStartTime : DTL;          // Cycle start timestamp

        // Last cycle summary
        // 0=None, 1=OK, 2=NOK, 3=STOP, 4=ABORT (Reset from an active state)
        LastResult     : Byte := 0;
        LastProgram    : Int := 0;
        LastDuration_s : DInt := 0;      // Duration in seconds
        LastErrorCode  : Word := 0;      // 0 if OK/STOP
        LastErrorLine  : Int := -1;      // -1 if not applicable
        LastEndTime    : DTL;            // End timestamp

        // NOTE (2026-07-31, memory reclaim): the 100-entry cycle history ring
        // (Hist_Index / Hist_Count / Hist_Result / Hist_Program / Hist_Duration_s /
        // Hist_ErrorCode / Hist_ErrorLine / Hist_Time) was removed -- it cost ~2.3 KB
        // of work memory but was write-only: nothing in the SCL ever read it back and
        // no HMI tag was mapped to it (see HMI_Tag_Guide.md).
        // The Total* counters and the last-cycle summary (Last*) are kept and remain the
        // HMI production source. (They were called "lifetime" counters here until
        // 2026-08-15, which was wrong at the time: the block was NON_RETAIN, so every
        // Total* zeroed on a power cycle. That keyword is now gone -- see the block
        // header -- but they only become genuinely lifetime once Retain is ticked per tag
        // in the TIA DB editor. Until then they still count per power-up.) Error-side history is unaffected --
        // DB_AlarmHistory (20 entries) and DB_Error.History_* still hold fault records.
        // To restore: re-add the arrays here and the push block in FB_Process
        // ("PRODUCTION LOGGING" section of 06_MainProcess.scl).
    END_VAR
BEGIN
END_DATA_BLOCK

// -----------------------------------------------------------------------------
// DB_fbSpindle -- FB_SpindleControl instance (NO LONGER CALLED IN OB1)
// Spindle is now controlled exclusively via fbSpindleControl inside FB_Process (fbProcess DB).
// This DB is retained so TIA Portal does not lose the symbol. Do not call from OB1.
// DB_Spindle (separate) → spindle status + HMI outputs (IsRunning, AtSpeed, etc.)
// -----------------------------------------------------------------------------
DATA_BLOCK "DB_fbSpindle"
{ S7_Optimized_Access := 'TRUE' }
VERSION : 0.1
NON_RETAIN
"FB_SpindleControl"
BEGIN
END_DATA_BLOCK

// =============================================================================
// PNEUMATIC CYLINDER INSTANCE DATA BLOCKS
// =============================================================================
// Instances of FBs defined in 09_Sensors_Actuators.scl.
// HMI reads/writes these DBs directly -- no separate interface DB needed.
//
// Cylinder map:
//   CylDiag[1] = DB_BackSupport    (full stroke, PositioningMode=0; ruler HW removed on this machine)
//   CylDiag[2] = DB_SheetHolder    (no sensor, PositioningMode=0, ValveType=2)
//   CylDiag[3] = DB_ToolHeadLock   (magnetic sensor, PositioningMode=1, safety lock)
//   CylDiag[4] = DB_MandrelLock    (no sensor, PositioningMode=0)
// =============================================================================

// =============================================================================
// BACKSUPPORT CYLINDER (CylDiag[1]) -- Full stroke, PositioningMode=0
//
// Ruler hardware removed on this machine. CMD=40 triggers a full extension;
// AtSetpoint fires after Timeout_Extend.
// DB_Cylinder_LinearRuler_BackSupport and OB1 ruler call are retained for future use
// if the ruler is re-fitted (switch PositioningMode back to 3 and re-enable in OB1).
// TIA tags:  Output_Cyl_Backsupport_SolA/B/Atmosphere
//
// COIL SEQUENCE (operator spec, 2026-08-07) -- the authority for this cylinder:
//
//   Event                     %Q12.0 Sol_A   %Q12.1 Sol_B   %Q12.7 Atmo
//   ------------------------- -------------- -------------- --------------
//   CMD=40                    ON (held)      off            off
//   CMD=41 P1                 ON (stays)     off            ON (held)
//   CMD=41 P2                 off            ON (retract)   off
//   CMD=41 P3                 off            off            off
//   Recipe end (any outcome)  off            ON 2s -> off   off
//
// Sol_A and Sol_B are NEVER energised together. Before 2026-08-07 they were:
// P1 also switched Sol_B on via an OR-override in OB1, and nothing ever released
// Sol_A (FB State 3 is a dead end for PositioningMode=0). The machine ran for
// months only because P1's wrong Sol_B happened to be the coil P2 needed, and
// Sol_B out-muscled the still-live Sol_A. That balance is pressure-dependent --
// when it tipped, the cylinder stopped retracting. See ITEM-41.
// =============================================================================

// -----------------------------------------------------------------------------
// DB_BackSupport -- FB_CylinderControl instance
// PositioningMode=0 (full stroke, timed), ValveType=2 (5/3 blocked center)
//
// HMI WRITABLE:   Cmd_ExtendFull, Cmd_RetractFull
// HMI READ-ONLY:  Sol_A, Sol_B, State, StateText, AtSetpoint, Error, ErrorID
// CONNECTED IN OB1: SafetyOK, RulerValue, RulerValid (ruler inputs ignored in Mode=0)
// To re-enable ruler: change PositioningMode to 3 and restore ruler tuning fields below.
// -----------------------------------------------------------------------------
DATA_BLOCK "DB_Cylinder_BackSupport"
{ S7_Optimized_Access := 'TRUE' }
VERSION : 0.5
NON_RETAIN
"FB_CylinderControl"
BEGIN
    ValveType           := 2;           // 5/3 blocked center -- mechanical lock in hold
    PositioningMode     := 0;           // Full stroke: extend on Cmd_Extend, AtSetpoint after Timeout_Extend
    Timeout_Extend      := T#3S;        // Measured extend stroke ~2s + margin. Was T#1S500MS, which was
                                        // SHORTER than the real stroke: STATE_CYL_GOTO_WAIT(71) advanced
                                        // mid-travel and CMD=41 P1 fired into a still-moving cylinder.
    Timeout_Retract     := T#24H;       // DELIBERATE -- do NOT shorten without measuring first.
                                        // The retract is commanded by CMD=41 P2 (Cmd_Retract latched)
                                        // and released by P3, so the window is RECIPE-controlled and
                                        // its upper bound has never been measured. While Cmd_Retract
                                        // is held the FB must stay in State 2 (Sol_A=FALSE, Sol_B=TRUE);
                                        // a timeout expiring mid-sequence would quietly stop driving
                                        // the cylinder back part-way through a P2..P3 window.
                                        // NOTE (2026-08-09): the old reason for this value is gone --
                                        // State 4 no longer latches Sol_B for Mode 0 + 5/3, it drives
                                        // both coils off like every other cylinder. Expiring is
                                        // therefore no longer dangerous, just premature. Once the real
                                        // P2..P3 duration is known this can become a normal timeout.
END_DATA_BLOCK

DATA_BLOCK "DB_Cylinder_Sen_BackSupport_Setpt"
{ S7_Optimized_Access := 'TRUE' }
VERSION : 0.1
NON_RETAIN
"FB_DigitalSensor"
BEGIN
    IsNC         := FALSE;
    DebounceTime := T#10ms;
END_DATA_BLOCK

// -----------------------------------------------------------------------------
// DB_Cylinder_LinearRuler_BackSupport -- FB_AnalogSensor instance
// Analog linear ruler for BackSupport cylinder position feedback.
// Connected in OB1: AI_LinearRuler_BackSupport → RulerValue/RulerValid on cylinder FB.
// Calibration is set in FC_LoadConfig Section 6; HMI can adjust at runtime.
// InvertSignal=TRUE: 0V = full extend (~300mm), ~10V = retracted (0mm).
// -----------------------------------------------------------------------------
DATA_BLOCK "DB_Cylinder_LinearRuler_BackSupport"
{ S7_Optimized_Access := 'TRUE' }
VERSION : 0.1
NON_RETAIN
"FB_AnalogSensor"
BEGIN
    Raw_Min      := 0;
    Raw_Max      := 31433;      // Measured at full retract -- update after hardware calibration
    Phys_Min     := 0.0;
    Phys_Max     := 300.0;      // Full stroke (mm) -- update if stroke differs
    InvertSignal := TRUE;       // 0V = extended end, ~10V = retracted end
    Hi_Limit     := 295.0;
    Lo_Limit     := 5.0;
END_DATA_BLOCK

// =============================================================================
// SHEETHOLDER CYLINDER (CylDiag[2]) -- No sensor, full stroke (PositioningMode=0)
//
// TIA Portal tags: Output_Cyl_SheetHolder_SolA (extend), Output_Cyl_SheetHolder_SolB (retract)
// Converted from 5/2 spring return to 5/3 blocked centre 2026-08-07 -- Sol_B is now wired.
// =============================================================================

// -----------------------------------------------------------------------------
// DB_SheetHolder -- FB_CylinderControl instance
// ValveType=2 (5/3 blocked centre, twin solenoid):
//   Sol_A=TRUE  → piston extends (sheet held).
//   Sol_B=TRUE  → piston retracts (active -- there is no spring any more).
//   Both FALSE  → blocked centre, piston mechanically locked where it stands.
//   Power loss  → both coils drop → piston LOCKED IN PLACE, it does NOT retract.
// PositioningMode=0: no sensor -- full stroke, timeout = done, no error.
//
// CONSEQUENCE FOR FB_PROCESS: the retract command must be HELD, not pulsed.
// With the old 5/2 the spring did the work, so a one-scan Cmd_Retract pulse was
// enough to kick the FB out of State 3. A one-scan pulse on a blocked centre
// energises Sol_B for a single scan and leaves the piston locked mid-stroke.
// FB_Process therefore holds Cmd_Retract via #bSheetHolderRetractHold for exactly
// DB_MachineConfig.CylSheetHolder_RetractTime, then drops it so BOTH coils
// de-energise and the blocked centre holds the piston at the retract end.
// See 06_MainProcess.scl "SHEETHOLDER COMMANDS -- single writer for BOTH directions".
// -----------------------------------------------------------------------------
DATA_BLOCK "DB_Cylinder_SheetHolder"
{ S7_Optimized_Access := 'TRUE' }
VERSION : 0.3
NON_RETAIN
"FB_CylinderControl"
BEGIN
    ValveType       := 2;       // 5/3 blocked centre -- twin solenoid, active retract on Sol_B
    PositioningMode := 0;       // No sensor -- full stroke, timeout = done, no error
    Timeout_Extend  := T#5S;
    // Backstop only -- it is NOT what ends the retract.
    //
    // The retract duration is owned by FB_Process: it holds Cmd_Retract for
    // DB_MachineConfig.CylSheetHolder_RetractTime (T#1S) and then drops it, which takes
    // the FB from State 2 to State 0 with both coils off. This value only decides what
    // happens if a retract is ever commanded for LONGER than that -- the FB gives up
    // waiting, calls the stroke done and moves to State 4, which since 2026-08-09 also
    // drives both coils off. So either exit ends with the coil de-energised and the
    // blocked centre holding the piston; the difference is cosmetic.
    //
    // (History: this was T#24H for a few hours during the ITEM-46 work, to dodge the old
    // State 4 behaviour where Mode 0 + 5/3 latched Sol_B ON for ever. That latch has been
    // deleted from FB_CylinderControl, so the dodge is no longer needed and a plain,
    // readable timeout is back. Keep it comfortably above CylSheetHolder_RetractTime.)
    Timeout_Retract := T#5S;
END_DATA_BLOCK

// =============================================================================
// TOOLHEADLOCK CYLINDER (CylDiag[3]) -- Magnetic sensor (PositioningMode=1, safety lock)
//
// LOCK BEHAVIOR (implemented in FB_Process):
//   EXTEND (Sol_A ON)  : states STATE_RUNNING (20) and STATE_PAUSED (25) only.
//   RETRACT (spring)   : all other states -- power loss also retracts (spring return).
//
// SEQUENCE GATES (FB_Process checks sensor before state transition):
//   Before entering RUNNING     : STATE_LOCK_EXTEND_WAIT (17) -- AtSetpoint OR 2s timer fallback.
//   Before TOOL_CHANGE / homing : STATE_LOCK_RETRACT_WAIT (29) -- 2s timer (no retract sensor).
//
// TIA Portal tags: In_Cyl_ToolHeadLock_AtSetpoint, Output_Cyl_ToolHeadLock_SolA
//                  (Sol_B not wired -- ValveType=1)
// =============================================================================

// -----------------------------------------------------------------------------
// DB_ToolHeadLock -- FB_CylinderControl instance
// ValveType=1 (5/2 spring return, single solenoid):
//   Sol_A=TRUE  → piston extends (locked).
//   Sol_A=FALSE → spring retracts (unlocked). Power loss = safe retract.
// Sen_AtSetpoint confirms lock fully engaged; Timeout_Extend=T#6S is error fallback.
// State 17 in FB_Process transitions when AtSetpoint=TRUE (sensor only; no fallback timer in FB_Process).
// Timeout_Extend in this DB is the only timer -- if sensor does not confirm within 6s, CylFB reports Error.
// -----------------------------------------------------------------------------
DATA_BLOCK "DB_Cylinder_ToolHeadLock"
{ S7_Optimized_Access := 'TRUE' }
VERSION : 0.3
NON_RETAIN
"FB_CylinderControl"
BEGIN
    ValveType       := 1;       // 5/2 spring return -- single solenoid, safe retract on power loss
    PositioningMode := 1;       // Mode 1: magnetic sensor -- AtSetpoint confirms lock engaged
    Timeout_Extend  := T#6S;    // Error 16#0501 if sensor not triggered within 6s of Cmd_Extend (raised from T#3S -- margin for slow pneumatic startup)
    Timeout_Retract := T#2S;    // Spring handles retract; timeout kept for completeness
END_DATA_BLOCK

DATA_BLOCK "DB_Cylinder_Sen_ToolHeadLock_Setpt"
{ S7_Optimized_Access := 'TRUE' }
VERSION : 0.1
NON_RETAIN
"FB_DigitalSensor"
BEGIN
    IsNC         := FALSE;
    DebounceTime := T#10ms;
END_DATA_BLOCK

// =============================================================================
// MANDRELLOCK CYLINDER (CylDiag[4]) -- No sensor, full stroke (PositioningMode=0)
//
// TIA Portal tags: Output_Cyl_MandrelLock_SolA, Output_Cyl_MandrelLock_SolB
// =============================================================================

// -----------------------------------------------------------------------------
// DB_MandrelLock -- FB_CylinderControl instance
// -----------------------------------------------------------------------------
DATA_BLOCK "DB_Cylinder_MandrelLock"
{ S7_Optimized_Access := 'TRUE' }
VERSION : 0.1
NON_RETAIN
"FB_CylinderControl"
BEGIN
    ValveType       := 1;       // 5/2
    PositioningMode := 0;       // No sensor -- full stroke, timeout = done, no error
    Timeout_Extend  := T#5S;
    Timeout_Retract := T#5S;
END_DATA_BLOCK

// -----------------------------------------------------------------------------
// DB_AlarmHistory - 20-entry alarm ring buffer for HMI history table (ITEM-26)
// NON_RETAIN: cleared on PLC power cycle. Survives Cmd_Reset (soft reset).
// HMI: connect Hist_Log[0..19] to a table, poll Hist_SeqNum for change detection,
//      sort by Timestamp descending. Hist_Clear = TRUE wipes manually.
// -----------------------------------------------------------------------------
DATA_BLOCK "DB_AlarmHistory"
{ S7_Optimized_Access := 'TRUE' }
VERSION : 0.1
NON_RETAIN
    VAR
        Hist_Head   : Int  := 0;       // Next write slot (0..19, wraps on overflow)
        Hist_Count  : Int  := 0;       // Number of valid entries (0..20)
        Hist_SeqNum : DInt := 0;       // Monotonically increasing — HMI polls for change detection
        Hist_Clear  : Bool := FALSE;   // HMI writes TRUE to clear history; auto-resets next scan
        Hist_Log    : Array[0..19] of "AlarmEntry";
    END_VAR
BEGIN
END_DATA_BLOCK

// -----------------------------------------------------------------------------
// DB_SelectedRecipe - the ONE recipe buffer the machine actually runs from
//                     (load-memory recipes, 2026-08-04)
//
// DB_RecipeProgram1..50 live in LOAD memory (UNLINKED) and cost no work memory.
// FB_RecipeLoader copies the selected one into here with READ_DBL during
// STATE_RECIPE_LOAD(11), before the pre-scan. FB_RecipePreScan and
// FB_RecipeHandler are then bound to THIS block and nothing else.
//
// { S7_Optimized_Access := 'FALSE' } is MANDATORY, not a style choice:
//   - READ_DBL requires source and destination to share a block access type,
//     and the recipe DBs must be standard (an optimized DB may not contain a
//     STRUCT, and RecipeLine is a UDT).
//   - Change it to 'TRUE' and every recipe load fails at runtime with 16#0312.
//
// This block must NEVER get the UNLINKED / "only store in load memory"
// attribute -- it is the destination, and it has to be readable by the program.
//
// Array bound must stay identical to DB_RecipeProgram*. Work memory cost:
// ~12 KB total, replacing the ~21 KB the five old work-memory recipe DBs used.
// See Program/docs/LOADMEM_COPY_ON_SELECT.md
// -----------------------------------------------------------------------------
DATA_BLOCK "DB_SelectedRecipe"
{ S7_Optimized_Access := 'FALSE' }
VERSION : 0.1
NON_RETAIN
    VAR
        Header : "RecipeHeader";                // Copy of the selected recipe's header
        // EXPERIMENTAL BOUND (branch exp/velocity-path-350, user decision 2026-09-14).
        // Was Array[0..999] with a "do not shrink" rule (2026-08-10): production parts
        // use ~1000 lines. Shrunk to 400 on this branch only (2026-09-14), raised to
        // 500 on 2026-09-16, to free work memory for the velocity-mode path experiment;
        // the 999-line parts need a coarser CAM export to run here. 500 still frees
        // ~11.7 KB against the 1000-line layout. Coupled change -- these move together
        // or READ_DBL fails on a length mismatch: LINES_PER_RECIPE / CHUNK_LINES in
        // tools/gen_recipe_slots.py, the two Lines InOuts in 05_RecipeHandler.scl,
        // the pre-scan guard (06_MainProcess.scl, activeLineCount > 500) and the
        // SpinningCam output.
        Lines  : Array[0..499] of "RecipeLine"; // Copy of the selected recipe's lines
    END_VAR
BEGIN
END_DATA_BLOCK

